{attribute addProperty BoxType "EP4374-0002-0016"}
{attribute addProperty Id "Analog_outputAT %Q*INT162"}
{attribute addProperty CRC "4118783225"}
{attribute addProperty SizeInBites "16"}
{attribute addProperty SizeInBytes "2"}
TYPE AO_RxPDO_Map_Channel_F57FA4F9 :
STRUCT
	{attribute addProperty Name "Analog_output"}
	Analog_output AT %Q* : INT;
END_STRUCT
END_TYPE

(* stored: Version 1.2.0.0, ProductVersion 3.1.4024.9
   DUT AO_RxPDO_Map_Channel_F57FA4F9: Id {e9b55212-0041-4a6e-afb3-d768ef84dc00} *)
